FUNCTION_BLOCK VariableToEvent (* Basic Function Block Type *)
  (* Standard: 61499-2 *)
  (* Version 0.2, 2003-12-04, JHC, Rockwell Automation, Renamed for better indexing. *)
  (* Version 0.1, 2002-11-05, JHC, Rockwell Automation, Corrected missing ST element in Algorithm REQ. *)
  (* Version 0.0, 2000-05-30, JHC, Rockwell Automation *)
  (* Compiler header: package fb.rt.cs725; *)
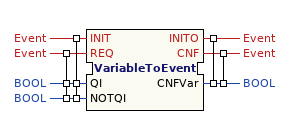
  EVENT_INPUT
    INIT WITH QI, NOTQI; (* Initialization Request *)
    REQ WITH QI, NOTQI; (* Normal Execution Request *)
  END_EVENT
  EVENT_OUTPUT
    INITO WITH CNFVar; (* Initialization Confirm *)
    CNF WITH CNFVar; (* Execution Confirmation *)
  END_EVENT
  VAR_INPUT
    QI : BOOL; (* Input event qualifier *)
    NOTQI : BOOL;
  END_VAR
  VAR_OUTPUT
    CNFVar : BOOL;
  END_VAR
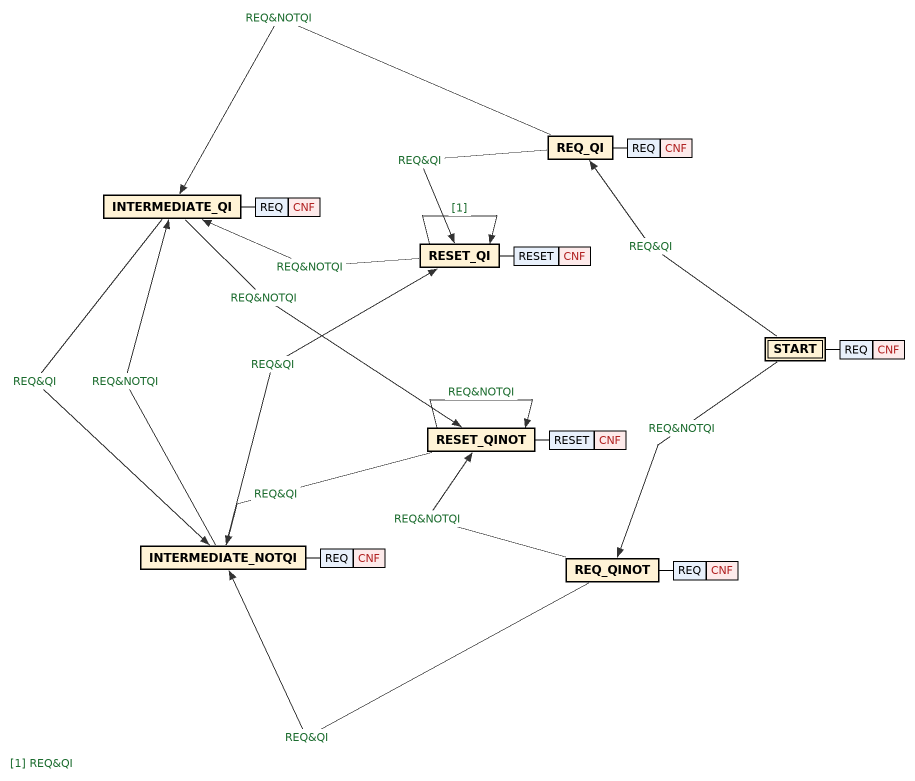
  EC_STATES
    START : REQ -> CNF; (* Initial State *)
    REQ_QI : REQ -> CNF; (* Normal execution *)
    RESET_QINOT : RESET -> CNF;
    REQ_QINOT : REQ -> CNF;
    RESET_QI : RESET -> CNF;
    INTERMEDIATE_QI : REQ -> CNF;
    INTERMEDIATE_NOTQI : REQ -> CNF;
  END_STATES
  EC_TRANSITIONS
    START TO REQ_QI := REQ&QI;
    START TO REQ_QINOT := REQ&NOTQI;
    REQ_QI TO RESET_QI := REQ&QI;
    REQ_QINOT TO RESET_QINOT := REQ&NOTQI;
    RESET_QI TO RESET_QI := REQ&QI;
    RESET_QINOT TO RESET_QINOT := REQ&NOTQI;
    REQ_QI TO INTERMEDIATE_QI := REQ&NOTQI;
    REQ_QINOT TO INTERMEDIATE_NOTQI := REQ&QI;
    INTERMEDIATE_NOTQI TO INTERMEDIATE_QI := REQ&NOTQI;
    INTERMEDIATE_QI TO INTERMEDIATE_NOTQI := REQ&QI;
    INTERMEDIATE_NOTQI TO RESET_QI := REQ&QI;
    INTERMEDIATE_QI TO RESET_QINOT := REQ&NOTQI;
    RESET_QI TO INTERMEDIATE_QI := REQ&NOTQI;
    RESET_QINOT TO INTERMEDIATE_NOTQI := REQ&QI;
  END_TRANSITIONS
  ALGORITHM INIT IN Java: (* Initialization algorithm *)
CNFVar.value = true;
  END_ALGORITHM
  ALGORITHM REQ IN Java: (* Normally executed algorithm *)
CNFVar.value = true;
System.out.println(this + "                  PE CHANGED!!!");
  END_ALGORITHM
  ALGORITHM RESET IN Java:
CNFVar.value=false;
System.out.println(this+"                            PE RESET/NOT CHANGED!!!");
  END_ALGORITHM
END_FUNCTION_BLOCK
